{attribute 'qualified_only'}
{attribute 'TcHmiSymbol' := 'true'}
VAR_GLOBAL
	
	bStartWrite : BOOL;
	bGeneratePDF: BOOL;
	bGeneratePDF2: BOOL;
	bStartRead: BOOL;
	bPreview: BOOL;
	localPDF : STRING;
	testPath : T_MaxString;
	sJsonOutput: STRING(100000);
	stReportHead: ST_ReportInfo;
	
(***** SQL Commands ***********************************************************************************)

//RUN CMDS	
isrtRun: STRING(5000) := 'INSERT INTO [dbo].[RUNS] ( [analyst], [comment], [softwareVersion], [sysMasterRevision], [sysSettingsRevision], [meterVelocity], [runVelocity], [emptyTubesFactor], [fillTubesFactor], [solvent1NameRevision], [solvent2NameRevision], [solvent3NameRevision], [solvent4NameRevision], [timeEventStarted], [timeEventCompleted], [methodID], [CalibrationNo]) VALUES ( $'#1#$', $'#2#$', $'#3#$', $'#4#$', $'#5#$', $'#6#$', $'#7#$', $'#8#$', $'#9#$', $'#10#$', $'#11#$', $'#12#$', $'#13#$', $'#14#$', $'#15#$', #16#, #17#) ';
slctLastRun: STRING(1000) := 'SELECT TOP 1 [runNo], [analyst], [comment], [softwareVersion], [sysMasterRevision], [sysSettingsRevision], [meterVelocity], [runVelocity], [emptyTubesFactor], [fillTubesFactor], [solvent1NameRevision], [solvent2NameRevision], [solvent3NameRevision], [solvent4NameRevision], [timeEventStarted], [timeEventCompleted], [methodID], [CalibrationNo] FROM [dbo].[RUNS] ORDER BY [runNo] DESC;';
//METHOD CMDS
slctAllMethods: STRING(5000) := 'SELECT [methodName], [methodRevision] FROM [dbo].[METHODS] ';
slctAllActvMethod: STRING(5000) := 'SELECT [methodName], [methodRevision] FROM [dbo].[METHODS] WHERE [methodStatus] = $'activated$'';
slctMethod: STRING(5000) := 'SELECT [methodName], [methodRevision], [methodCreatedBy], [methodCreatedOn], [solvent_R1], [solvent_R2], [solvent_W1], [solvent_W2], [time_R1], [time_R2], [time_W1], [time_W2], [velocity_R1], [velocity_R2], [velocity_W1], [velocity_W2], [soakTime], [agitate_1_Time], [agitate_2_Time], [vialsToFill], [vialPrimeVol], [vial_1_FillVol], [vial_2_4_FillVol], [airDryTime], [methodID], [methodStatus] FROM [dbo].[METHODS] WHERE [methodName] = $'#1#$' AND [methodRevision] = $'#2#$' ';
slctVD: STRING(5000) := 'SELECT [VD_ID], [pump], [stage], [rinse1], [rinse2], [wash1], [wash2], [methodID] FROM [dbo].[VOLUME_DATA] WHERE [methodID] = #1# ';
isrtNewMethod: STRING(5000) := 'INSERT INTO [dbo].[METHODS] ( [methodName], [methodRevision], [methodCreatedBy], [methodCreatedOn], [solvent_R1], [solvent_R2], [solvent_W1], [solvent_W2], [time_R1], [time_R2], [time_W1], [time_W2], [velocity_R1], [velocity_R2], [velocity_W1], [velocity_W2], [soakTime], [agitate_1_Time], [agitate_2_Time], [vialsToFill], [vialPrimeVol], [vial_1_FillVol], [vial_2_4_FillVol], [airDryTime], [methodStatus]) VALUES ( $'#1#$', $'#2#$', $'#3#$', $'#4#$', $'#5#$', $'#6#$', $'#7#$', $'#8#$', $'#9#$', $'#10#$', $'#11#$', $'#12#$', $'#13#$', $'#14#$', $'#15#$', $'#16#$', $'#17#$', $'#18#$', $'#19#$', $'#20#$', $'#21#$', $'#22#$', $'#23#$', $'#24#$', $'#25#$') ';
isrtVD: string(5000) := 'INSERT INTO [dbo].[VOLUME_DATA] ( [pump], [stage], [rinse1], [rinse2], [wash1], [wash2], [methodID]) VALUES ( $'#1#$', $'#2#$', $'#3#$', $'#4#$', $'#5#$', $'#6#$', #7#) ';
updtDactvMethod: STRING(5000) := 'UPDATE [dbo].[METHODS] SET [methodStatus] = $'deactivated$' WHERE [methodName] = $'#1#$' AND [methodRevision] = $'#2#$'';
//CALIBRATION CMD
slctLastCalibID: T_Maxstring := 'SELECT TOP 1 [calibrationNo] FROM [dbo].[CALIBRATION] ORDER BY [calibrationNo] DESC;';
isrtCalib: STRING(5000) := 'INSERT INTO [dbo].[CALIBRATION_HEAD] ( [userID], [density], [solventNo], [solventRevision], [allowableFail], [replicates], [callInterval], [sysRevisionNo]) VALUES ( $'#1#$', $'#2#$', $'#3#$', $'#4#$', $'#5#$', $'#6#$', $'#7#$', #8#) ';
isrtCalibValues: STRING(5000) := 'INSERT INTO [dbo].[CALIBRATION] ( [dateTime], [pumpNo], [step], [tareWt], [grossWt], [netVolume], [netWt], [targetVolume], [differencePercent], [criteria], [pumpRevs], [CalibrationNo]) VALUES ( $'#1#$', $'#2#$', $'#3#$', $'#4#$', $'#5#$', $'#6#$', $'#7#$', $'#8#$', $'#9#$', $'#10#$', $'#11#$', #12#) ';
//SYSTEM CMD
slctLastSys: STRING(5000) := 'SELECT TOP 1 [gen_SealAndPump], [cal_AcceptanceCriteria], [cal_AllowableFail], [cal_Replicates], [cal_PumpCallIntervalDays], [cal_CloseAppOnCompletation], [AirDryTimeOnCompletation], [lkt_AllowableLeakTestFail], [lkt_LeakTestBuildupTime], [lkt_LeakTestHoldTime], [lkt_LeakTestPressure], [mec_PlatesClosedPosition], [mec_PlatesDryPosition], [mec_PlatesVelocity], [mec_MaxCurrentFastDown], [mec_MaxCurrentSlowDown], [mec_MaxCurrentSlowUp], [pmp_MeterVelocity], [pmp_RunVelocity], [pmp_EmptyFactor], [pmp_FillSolventTubesFactor], [smp_AboveCalibration], [smp_VialSetSpacing], [smp_IntoResBottom], [smp_IntoResDispense], [smp_IntoResWeigh], [smp_IntoVials], [sec_DisplayManualControl], [sec_CheckLogonEachRun], [createdBy], [createdDate], [sysRevisionNo] FROM [dbo].[SYSTEM] ORDER BY [sysRevisionNo] DESC; ';
isrtSys: STRING(5000) := 'INSERT INTO [dbo].[SYSTEM] ( [gen_SealAndPump], [cal_AcceptanceCriteria], [cal_AllowableFail], [cal_Replicates], [cal_PumpCallIntervalDays], [cal_CloseAppOnCompletation], [AirDryTimeOnCompletation], [lkt_AllowableLeakTestFail], [lkt_LeakTestBuildupTime], [lkt_LeakTestHoldTime], [lkt_LeakTestPressure], [mec_PlatesClosedPosition], [mec_PlatesDryPosition], [mec_PlatesVelocity], [mec_MaxCurrentFastDown], [mec_MaxCurrentSlowDown], [mec_MaxCurrentSlowUp], [pmp_MeterVelocity], [pmp_RunVelocity], [pmp_EmptyFactor], [pmp_FillSolventTubesFactor], [smp_AboveCalibration], [smp_VialSetSpacing], [smp_IntoResBottom], [smp_IntoResDispense], [smp_IntoResWeigh], [smp_IntoVials], [sec_DisplayManualControl], [sec_CheckLogonEachRun], [createdBy], [createdDate]) VALUES ( $'#1#$', $'#2#$', $'#3#$', $'#4#$', $'#5#$', $'#6#$', $'#7#$', $'#8#$', $'#9#$', $'#10#$', $'#11#$', $'#12#$', $'#13#$', $'#14#$', $'#15#$', $'#16#$', $'#17#$', $'#18#$', $'#19#$', $'#20#$', $'#21#$', $'#22#$', $'#23#$', $'#24#$', $'#25#$', $'#26#$', $'#27#$', $'#28#$', $'#29#$', $'#30#$', $'#31#$') ';
//USERS CMD
isrtUser: STRING(5000) := 'INSERT INTO [dbo].[USERS] ( [userID], [acessLevel], [transactionType], [transactionDate], [transactedBy], [addDate], [enteredBy]) VALUES ( $'#1#$', $'#2#$', $'#3#$', $'#4#$', $'#5#$', $'#6#$', $'#7#$') ';
slctCurrentUser: STRING(5000) := 'SELECT [ID_user], [userID], [acessLevel], [transactionType], [transactionDate], [transactedBy], [addDate], [enteredBy] FROM [dbo].[USERS] u WHERE [transactionType] = $'Added$' AND [transactionDate] = (SELECT MAX([transactionDate]) FROM [dbo].[USERS] WHERE [userID] = u.[userID] AND [transactionType] = $'Added$')';//'SELECT [ID_user], [userID], [acessLevel], [transactionType], [transactionDate], [transactedBy], [addDate], [enteredBy] FROM [dbo].[USERS] u WHERE [transactionType] = $'Added$' AND [ID_user] = ( SELECT MAX([ID_user]) FROM [dbo].[USERS] WHERE [userID] = u.[userID] AND [transactionType] = $'Added$');';
slctAllUsers: STRING(5000) := 'SELECT [ID_user], [userID], [acessLevel], [transactionType], [transactionDate], [transactedBy], [addDate], [enteredBy] FROM [dbo].[USERS] ';


(******************************************************************************************************)

(***** Pump Calibration Report Variables **************************************************************)

bBuildPCR			: BOOL;
stParameter_PCR		: ST_Parameters_PCR;
astData_PCR	  		: ARRAY[0..100] OF ST_Data_PCR;
lastCalibID			: ARRAY[0..1] OF INT;


(******************************************************************************************************)
	
(***** Post-Run Report Variables **********************************************************************)

bBuildPRRW		: BOOL;
stPostRunReport	: ARRAY[0..5] OF ST_PostRunReport;
lastRunID		: ARRAY[0..1] OF INT;

(******************************************************************************************************)

(***** User History Report Variables ******************************************************************)

bBuildUHR	   : BOOL;
astData_UHR	   : ARRAY[0..100] OF ST_Data_UHR;

(******************************************************************************************************)

(***** Current Users List Variables *****************************************************************)

bBuildCUL	   : BOOL;
astData_CUL	   : ARRAY[0..1000] OF ST_Data_CUL;

(******************************************************************************************************)

(***** Method Report Variables ************************************************************************)

bBuildMR		: BOOL;
stParameter_MR	: ST_Parameters_MR;
astVolData		: ARRAY[1..10] OF ST_VolumeData;
listOfMethod	: ARRAY[1..500] OF ST_ListMethod;

(******************************************************************************************************)

(***** System Parameters Variables ***************************************************************)

stSysParameters	: ARRAY[0..1] OF ST_SysParameters;

(******************************************************************************************************)

(***** System Settings History Report Variables *******************************************************)

(******************************************************************************************************)
END_VAR

(* stored: Version 1.1.0.1, ProductVersion 3.1.4024.15
   GVL GVL_DB: Id {b6405db0-d623-4e3b-8d34-c8eb4e42140d} *)
